// TIA Portal project "sıralı_lamp_toggle" (V18)

(* hardware
DEVICE "S7-1200 station_1"  S7-1200 Station
   slot 0: "Rack_0"  S7-1200 Rack  Rack  V1.0
   slot 1: "PLC_1"  CPU 1212C DC/DC/Rly  6ES7 212-1HE40-0XB0  V4.6
*)

// ===== PLC "PLC_1"  CPU 1212C DC/DC/Rly =====

VAR_GLOBAL   // PLC tag table "Default tag table"
   "B0" AT %M0.0 : Bool;
   "B1" AT %M0.1 : Bool;
   "B2" AT %M0.2 : Bool;
   "B3" AT %M0.3 : Bool;
   "BTN" AT %I0.0 : Bool;
   "M0" AT %M1.0 : Bool;
   "A1" AT %M2.0 : Bool;
   "A2" AT %M2.1 : Bool;
   "M1" AT %M1.1 : Bool;
   "A3" AT %M2.2 : Bool;
   "M2" AT %M1.2 : Bool;
   "L1" AT %Q0.0 : Bool;
   "L2" AT %Q0.1 : Bool;
   "L3" AT %Q0.2 : Bool;
   "L4" AT %Q0.3 : Bool;
END_VAR

FUNCTION "Block_1" : Void   // FC1, LAD
{ S7_Optimized_Access := 'TRUE' }
VERSION : 0.1
   VAR_TEMP   // added for the SCL form of the ladder/FBD networks
      _w1 : Bool;
   END_VAR
BEGIN

REGION Network 1
   // BIT0
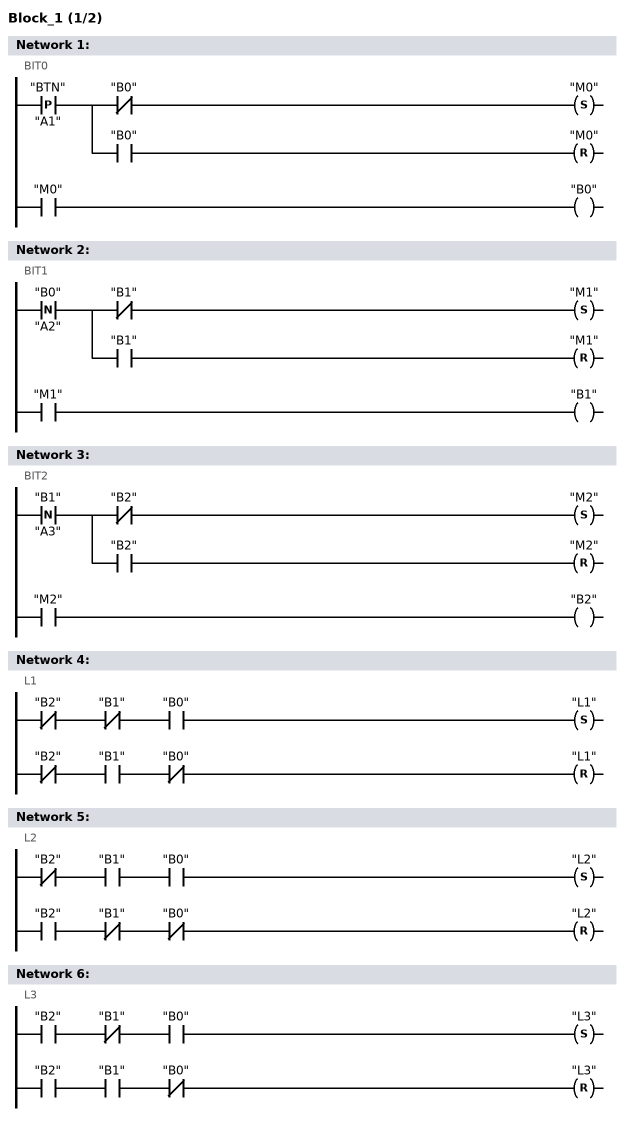
   RUNG wire#powerrail
      P_Contact(operand := "BTN", bit := "A1")
      wire#w1
      I_Contact( "B0" )
      S_Coil( "M0" )
   END_RUNG
   RUNG wire#w1
      Contact( "B0" )
      R_Coil( "M0" )
   END_RUNG
   RUNG wire#powerrail
      Contact( "M0" )
      Coil( "B0" )
   END_RUNG
   // the same network as SCL:
   #_w1 := "BTN" AND NOT "A1";   // rising edge of "BTN"
   "A1" := "BTN";
   IF #_w1 AND NOT "B0" THEN "M0" := TRUE; END_IF;
   IF #_w1 AND "B0" THEN "M0" := FALSE; END_IF;
   "B0" := "M0";
END_REGION

REGION Network 2
   // BIT1
   RUNG wire#powerrail
      N_Contact(operand := "B0", bit := "A2")
      wire#w1
      I_Contact( "B1" )
      S_Coil( "M1" )
   END_RUNG
   RUNG wire#w1
      Contact( "B1" )
      R_Coil( "M1" )
   END_RUNG
   RUNG wire#powerrail
      Contact( "M1" )
      Coil( "B1" )
   END_RUNG
   // the same network as SCL:
   #_w1 := NOT "B0" AND "A2";   // falling edge of "B0"
   "A2" := "B0";
   IF #_w1 AND NOT "B1" THEN "M1" := TRUE; END_IF;
   IF #_w1 AND "B1" THEN "M1" := FALSE; END_IF;
   "B1" := "M1";
END_REGION

REGION Network 3
   // BIT2
   RUNG wire#powerrail
      N_Contact(operand := "B1", bit := "A3")
      wire#w1
      I_Contact( "B2" )
      S_Coil( "M2" )
   END_RUNG
   RUNG wire#w1
      Contact( "B2" )
      R_Coil( "M2" )
   END_RUNG
   RUNG wire#powerrail
      Contact( "M2" )
      Coil( "B2" )
   END_RUNG
   // the same network as SCL:
   #_w1 := NOT "B1" AND "A3";   // falling edge of "B1"
   "A3" := "B1";
   IF #_w1 AND NOT "B2" THEN "M2" := TRUE; END_IF;
   IF #_w1 AND "B2" THEN "M2" := FALSE; END_IF;
   "B2" := "M2";
END_REGION

REGION Network 4
   // L1
   RUNG wire#powerrail
      I_Contact( "B2" )
      I_Contact( "B1" )
      Contact( "B0" )
      S_Coil( "L1" )
   END_RUNG
   RUNG wire#powerrail
      I_Contact( "B2" )
      Contact( "B1" )
      I_Contact( "B0" )
      R_Coil( "L1" )
   END_RUNG
   // the same network as SCL:
   IF NOT "B2" AND NOT "B1" AND "B0" THEN "L1" := TRUE; END_IF;
   IF NOT "B2" AND "B1" AND NOT "B0" THEN "L1" := FALSE; END_IF;
END_REGION

REGION Network 5
   // L2
   RUNG wire#powerrail
      I_Contact( "B2" )
      Contact( "B1" )
      Contact( "B0" )
      S_Coil( "L2" )
   END_RUNG
   RUNG wire#powerrail
      Contact( "B2" )
      I_Contact( "B1" )
      I_Contact( "B0" )
      R_Coil( "L2" )
   END_RUNG
   // the same network as SCL:
   IF NOT "B2" AND "B1" AND "B0" THEN "L2" := TRUE; END_IF;
   IF "B2" AND NOT "B1" AND NOT "B0" THEN "L2" := FALSE; END_IF;
END_REGION

REGION Network 6
   // L3
   RUNG wire#powerrail
      Contact( "B2" )
      I_Contact( "B1" )
      Contact( "B0" )
      S_Coil( "L3" )
   END_RUNG
   RUNG wire#powerrail
      Contact( "B2" )
      Contact( "B1" )
      I_Contact( "B0" )
      R_Coil( "L3" )
   END_RUNG
   // the same network as SCL:
   IF "B2" AND NOT "B1" AND "B0" THEN "L3" := TRUE; END_IF;
   IF "B2" AND "B1" AND NOT "B0" THEN "L3" := FALSE; END_IF;
END_REGION

REGION Network 7
   // L4
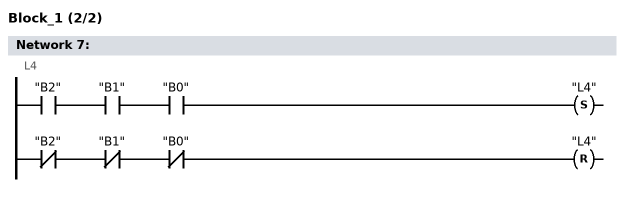
   RUNG wire#powerrail
      Contact( "B2" )
      Contact( "B1" )
      Contact( "B0" )
      S_Coil( "L4" )
   END_RUNG
   RUNG wire#powerrail
      I_Contact( "B2" )
      I_Contact( "B1" )
      I_Contact( "B0" )
      R_Coil( "L4" )
   END_RUNG
   // the same network as SCL:
   IF "B2" AND "B1" AND "B0" THEN "L4" := TRUE; END_IF;
   IF NOT "B2" AND NOT "B1" AND NOT "B0" THEN "L4" := FALSE; END_IF;
END_REGION
END_FUNCTION

ORGANIZATION_BLOCK "Main"   // OB1, LAD, ProgramCycle
TITLE = "Main Program Sweep (Cycle)"
{ S7_Optimized_Access := 'TRUE' }
VERSION : 0.1
   VAR_INPUT
      Initial_Call : Bool;   // Initial call of this OB
      Remanence : Bool;   // =True, if remanent data are available
   END_VAR
BEGIN

REGION Network 1
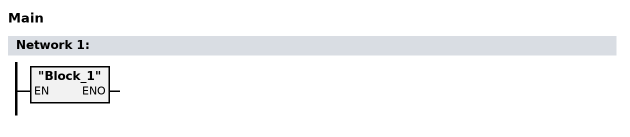
   RUNG wire#powerrail
      "Block_1"()
   END_RUNG
   // the same network as SCL:
   "Block_1"();
END_REGION
END_ORGANIZATION_BLOCK